KUKA KRL program: separa.src, separa.dat

--- separa.src ---
&ACCESS RV
DEF separa ( )

END

--- separa.dat ---
&ACCESS RV
DEFDAT separa PUBLIC

ENDDAT
